PROGRAM DB_Create_Calibration
VAR
	state: INT;
	timer: ton;
END_VAR

VAR_INPUT
	start: BOOL;
END_VAR

timer();

CASE state OF
	
0:
	IF start THEN
		DB_Query.state:= E_DB_QUERY_STATE.SELECT_LAST_CALIBRATION_ID;
		timer(in:=TRUE, pt:=T#10S);
		state:= 10;
	ELSE
		state:= 0;
	END_IF

10:

	IF NOT DB_Query.FB_SelectArray.bBusy AND timer.Q THEN
		timer(in:=FALSE);
		GVL_Calibration.stPumpCalibrationInfo.iCalibrationNumber 		:= GVL_DB.lastCalibID[0];	
		GVL_DB.stParameter_PCR.userID									:= 'DEV';
		GVL_DB.stParameter_PCR.allowableFail							:= USINT_TO_STRING(GVL_Settings.stCalibParameters.iAllowableFailures);
		GVL_DB.stParameter_PCR.CalibrationNo							:= UDINT_TO_INT(GVL_Calibration.stPumpCalibrationInfo.iCalibrationNumber+1);
		GVL_DB.stParameter_PCR.callInterval								:= UINT_TO_STRING(GVL_Settings.stCalibParameters.iCalIntervalDays);
		GVL_DB.stParameter_PCR.density									:= REAL_TO_STRING(GVL_Calibration.stPumpCalibrationInfo.rSolventDensity);
		GVL_DB.stParameter_PCR.replicates								:= INT_TO_STRING(GVL_Settings.stCalibParameters.iReplicatesSetpoint);
		GVL_DB.stParameter_PCR.solventNo								:= GVL_Calibration.stPumpCalibrationInfo.iSolventID;
		GVL_DB.stParameter_PCR.solventRevision							:= INT_TO_STRING(GVL_Calibration.stPumpCalibrationInfo.iSolventRevision);
		GVL_DB.stParameter_PCR.sysRevisionNo							:= GVL_Settings.sysRevNumber;	
		state:= 20;
	ELSE
		state:= 10;
	END_IF
	
20:

	IF TRUE THEN
		DB_Query.state:= E_DB_QUERY_STATE.INSERT_CALIBRATION;
		timer(in:=TRUE, pt:=T#10S);
		state:= 30;
	ELSE
		state:= 20;
	END_IF	

30:

	IF NOT DB_Query.FB_Insert.bBusy AND timer.Q THEN
		timer(in:=FALSE);
		start:= FALSE;
		state:= 0;
	ELSE
		state:= 30;
	END_IF
END_CASE

END_PROGRAM

(* stored: Version 1.1.0.1, ProductVersion 3.1.4024.15
   POU DB_Create_Calibration: Id {373c1b49-6b74-4b04-86ce-e0678f5d1ec2}, SpecialFunc None *)
